// Mitsubishi GX Works2 project: Fx3U_ModbusRTU   PLC: FX3U/FX3UC

PROGRAM MAIN
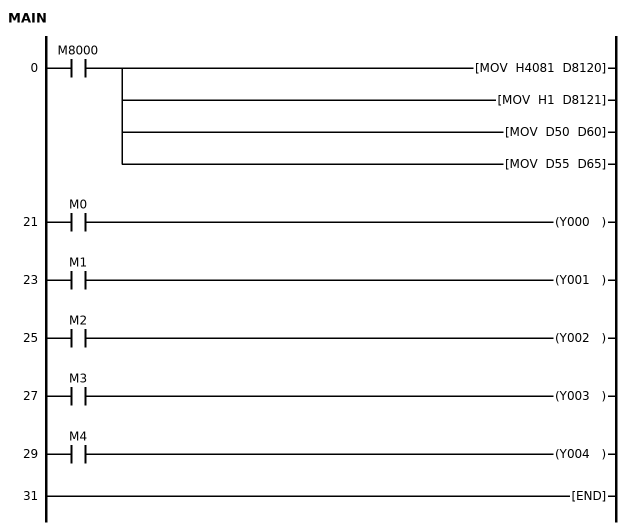
0     LD      M8000
      MOV     H4081 D8120
      MOV     H1 D8121
      MOV     D50 D60
      MOV     D55 D65
21    LD      M0
      OUT     Y000
23    LD      M1
      OUT     Y001
25    LD      M2
      OUT     Y002
27    LD      M3
      OUT     Y003
29    LD      M4
      OUT     Y004
31    END
END_PROGRAM
